// TIA Portal V16 export
FUNCTION_BLOCK "FB_Conveyor_LAD"   // FB2, LAD
{ S7_Optimized_Access := 'TRUE' }
// stored: AutoNumber false
   VAR_INPUT
      FirstScan : Bool;
      StartButton : Bool;
      StopOK : Bool;
      EStopOK : Bool;
      OverloadOK : Bool;
      JamSensor : Bool;
      ResetButton : Bool;
      JamTime : Time := T#5s;
   END_VAR
   VAR_OUTPUT
      MotorCmd : Bool;
      RunLamp : Bool;
      FaultLamp : Bool;
   END_VAR
   VAR
      RunLatch : Bool := FALSE;
      FaultLatch : Bool := FALSE;
      JamTimer : TON_TIME;
   END_VAR
BEGIN

REGION Network 1: 01 - First scan: reset run latch
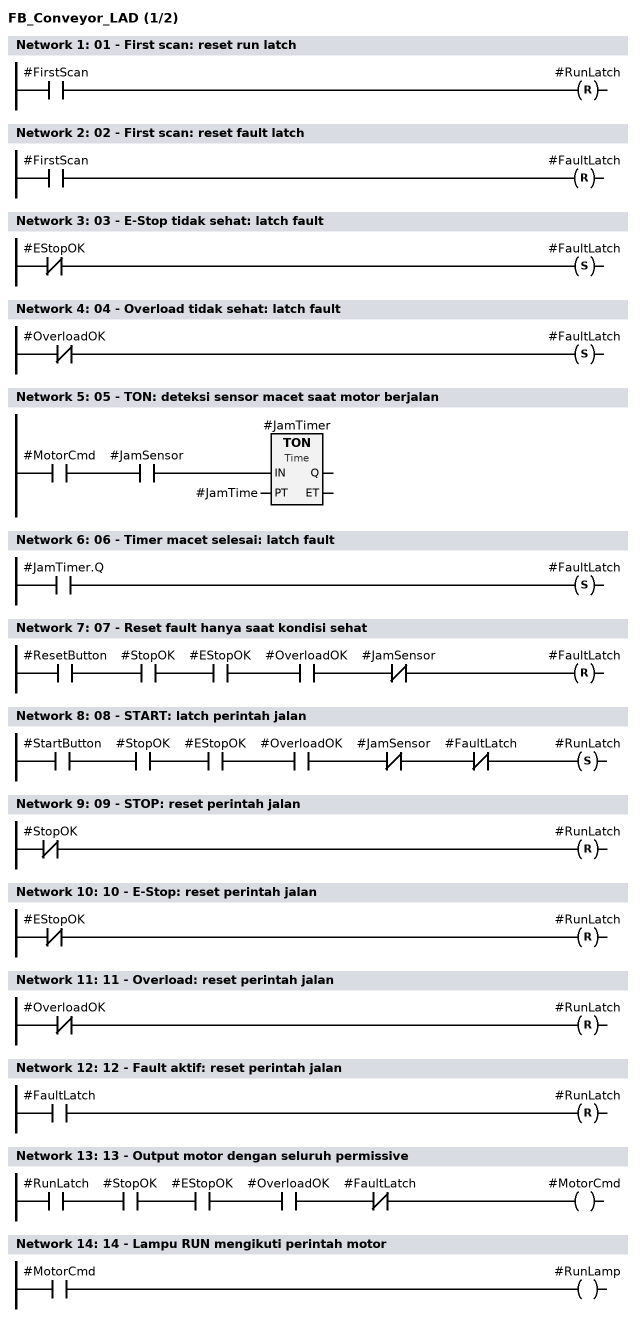
   RUNG wire#powerrail
      Contact( #FirstScan )
      R_Coil( #RunLatch )
   END_RUNG
   // the same network as SCL:
   IF #FirstScan THEN #RunLatch := FALSE; END_IF;
END_REGION

REGION Network 2: 02 - First scan: reset fault latch
   RUNG wire#powerrail
      Contact( #FirstScan )
      R_Coil( #FaultLatch )
   END_RUNG
   // the same network as SCL:
   IF #FirstScan THEN #FaultLatch := FALSE; END_IF;
END_REGION

REGION Network 3: 03 - E-Stop tidak sehat: latch fault
   RUNG wire#powerrail
      I_Contact( #EStopOK )
      S_Coil( #FaultLatch )
   END_RUNG
   // the same network as SCL:
   IF NOT #EStopOK THEN #FaultLatch := TRUE; END_IF;
END_REGION

REGION Network 4: 04 - Overload tidak sehat: latch fault
   RUNG wire#powerrail
      I_Contact( #OverloadOK )
      S_Coil( #FaultLatch )
   END_RUNG
   // the same network as SCL:
   IF NOT #OverloadOK THEN #FaultLatch := TRUE; END_IF;
END_REGION

REGION Network 5: 05 - TON: deteksi sensor macet saat motor berjalan
   RUNG wire#powerrail
      Contact( #MotorCmd )
      Contact( #JamSensor )
      { S7_Templates := "time_type := Time" } #JamTimer.TON(pt := #JamTime, et =>)
   END_RUNG
   // the same network as SCL:
   #JamTimer(IN := #MotorCmd AND #JamSensor, PT := #JamTime);   // TON
END_REGION

REGION Network 6: 06 - Timer macet selesai: latch fault
   RUNG wire#powerrail
      Contact( #JamTimer.Q )
      S_Coil( #FaultLatch )
   END_RUNG
   // the same network as SCL:
   IF #JamTimer.Q THEN #FaultLatch := TRUE; END_IF;
END_REGION

REGION Network 7: 07 - Reset fault hanya saat kondisi sehat
   RUNG wire#powerrail
      Contact( #ResetButton )
      Contact( #StopOK )
      Contact( #EStopOK )
      Contact( #OverloadOK )
      I_Contact( #JamSensor )
      R_Coil( #FaultLatch )
   END_RUNG
   // the same network as SCL:
   IF #ResetButton AND #StopOK AND #EStopOK AND #OverloadOK AND NOT #JamSensor THEN
       #FaultLatch := FALSE;
   END_IF;
END_REGION

REGION Network 8: 08 - START: latch perintah jalan
   RUNG wire#powerrail
      Contact( #StartButton )
      Contact( #StopOK )
      Contact( #EStopOK )
      Contact( #OverloadOK )
      I_Contact( #JamSensor )
      I_Contact( #FaultLatch )
      S_Coil( #RunLatch )
   END_RUNG
   // the same network as SCL:
   IF #StartButton AND #StopOK AND #EStopOK AND #OverloadOK AND NOT #JamSensor AND NOT #FaultLatch THEN
       #RunLatch := TRUE;
   END_IF;
END_REGION

REGION Network 9: 09 - STOP: reset perintah jalan
   RUNG wire#powerrail
      I_Contact( #StopOK )
      R_Coil( #RunLatch )
   END_RUNG
   // the same network as SCL:
   IF NOT #StopOK THEN #RunLatch := FALSE; END_IF;
END_REGION

REGION Network 10: 10 - E-Stop: reset perintah jalan
   RUNG wire#powerrail
      I_Contact( #EStopOK )
      R_Coil( #RunLatch )
   END_RUNG
   // the same network as SCL:
   IF NOT #EStopOK THEN #RunLatch := FALSE; END_IF;
END_REGION

REGION Network 11: 11 - Overload: reset perintah jalan
   RUNG wire#powerrail
      I_Contact( #OverloadOK )
      R_Coil( #RunLatch )
   END_RUNG
   // the same network as SCL:
   IF NOT #OverloadOK THEN #RunLatch := FALSE; END_IF;
END_REGION

REGION Network 12: 12 - Fault aktif: reset perintah jalan
   RUNG wire#powerrail
      Contact( #FaultLatch )
      R_Coil( #RunLatch )
   END_RUNG
   // the same network as SCL:
   IF #FaultLatch THEN #RunLatch := FALSE; END_IF;
END_REGION

REGION Network 13: 13 - Output motor dengan seluruh permissive
   RUNG wire#powerrail
      Contact( #RunLatch )
      Contact( #StopOK )
      Contact( #EStopOK )
      Contact( #OverloadOK )
      I_Contact( #FaultLatch )
      Coil( #MotorCmd )
   END_RUNG
   // the same network as SCL:
   #MotorCmd := #RunLatch AND #StopOK AND #EStopOK AND #OverloadOK AND NOT #FaultLatch;
END_REGION

REGION Network 14: 14 - Lampu RUN mengikuti perintah motor
   RUNG wire#powerrail
      Contact( #MotorCmd )
      Coil( #RunLamp )
   END_RUNG
   // the same network as SCL:
   #RunLamp := #MotorCmd;
END_REGION

REGION Network 15: 15 - Lampu FAULT mengikuti fault latch
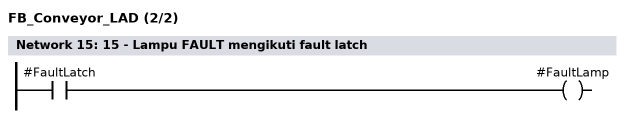
   RUNG wire#powerrail
      Contact( #FaultLatch )
      Coil( #FaultLamp )
   END_RUNG
   // the same network as SCL:
   #FaultLamp := #FaultLatch;
END_REGION
END_FUNCTION_BLOCK
